FUNCTION_BLOCK FINAL FB_Cylinder EXTENDS FB_EventLogger 
VAR_INPUT
	Energized						: BOOL;							//Optional Energize Input
END_VAR                                                     		
VAR_IN_OUT                                                  		
	Control							: ST_System;					//Machine Control Instance
END_VAR                                                     		
VAR                                                         		
	_AutoExtend						: BOOL;							//Automated Extend Signal
	_AutoRetract					: BOOL;							//Automated Retract Signal
	_ManExtend						: BOOL;							//Screen Selection
	_ManRetract						: BOOL;							//Screen Selection
	_ManOff							: BOOL;							//Screen Selection
	_ForceExtend					: BOOL;							//Screen Selection
	_ForceRetract					: BOOL;							//Screen Selection
	_ForceOff						: BOOL;							//Screen Selection
	_CycleEnable					: BOOL;							//Cylinder Cylce Enable
	_ExtendReed1		AT %I*		: BOOL;							//Cylinder Extend Reed 1
	_ExtendReed2		AT %I*		: BOOL;							//Cylinder Extend Reed 2
	_ExtendReed3		AT %I*		: BOOL;							//Cylinder Extend Reed 3
	_ExtendReed4		AT %I*		: BOOL;							//Cylinder Extend Reed 4
	_RetractReed1		AT %I*		: BOOL;							//Cylinder Retract Reed 1
	_RetractReed2		AT %I*		: BOOL;							//Cylinder Retract Reed 2
	_RetractReed3		AT %I*		: BOOL;							//Cylinder Retract Reed 3
	_RetractReed4		AT %I*		: BOOL;							//Cylinder Retract Reed 4
	_DualSolenoid					: BOOL;							//Configured as a dual Solenoid Device
	_SingleSolenoidNormal			: BOOL;							//Configured as a Signal Solenoid Extend Device (Default)	
	_SingleSolenoidReverse			: BOOL;							//Configured as a Signal Solenoid Retract Device
	_CountsReset					: BOOL;							//Cycle Counts Reset
	_CycleExtend					: BOOL;							//Cylinder Cycle Extend
	_CycleRetract					: BOOL;							//Cylinder Cycle Retract
	_ExtendSolOnTime_ET				: REAL;							//Time Extend Solenoid Has Been Energised
	_ExtendSolOffTime_ET			: REAL;							//Time Since Extend Solenoid was Last Energised
	_RetractSolOnTime_ET			: REAL;							//Time Retract Solenoid Has Been Energised
	_RetractSolOffTime_ET			: REAL;							//Time Since Retract Solenoid was Last Energised
	_ExtendTime_ET					: REAL;							//Time Cylinder has been Extended
	_RetractTime_ET					: REAL;							//Time Cylinder has been Retracted
	_CycleExtTime_ET				: REAL;							//Cylinder Cycle Extend Accumulated Time
	_CycleRetTime_ET				: REAL;							//Cylinder Cycle Retract Accumulated Time
	_ExtendReed						: BOOL;							//All cylinder extend reeds have been made
	_RetractReed					: BOOL;							//All cylinder retract reeds have been made
	_ReedFaultCount					: SINT;							//Count for type of reed fault
	_ExtendSol				AT %Q*	: BOOL;							//Physical output for extend solenoid
	_RetractSol				AT %Q*	: BOOL;							//Physical output for retract solenoid
	_ExtendFault					: BOOL;							//Fault for cylinder extend
	_RetractFault					: BOOL;							//Fault for cylinder retract
	_ReedFault						: BOOL;							//Fault for reed
	_ReedFaultTime_ET				: REAL;							//Reed fault elapsed time
	_ExFaultTime_ET					: REAL;							//Extend fault elapsed time
	_RtFaultTime_ET					: REAL;							//Retract fault elapsed time
	_Alarm							: BOOL;							//Device Alarm
	_Warning						: BOOL;							//Device Warning
	_AlarmNum						: DINT;							//Device Alarm Number
	_WarningNum						: DINT;							//Device Warning Number
	_Mute_Retract					: BOOL;							//Mute Retract Alarm
	_Mute_Extend					: BOOL;							//Mute Extend Alarm
	_extendReedUsed1				: BOOL;                 	
	_extendReedUsed2				: BOOL;                 	
	_extendReedUsed3				: BOOL;                 	
	_extendReedUsed4				: BOOL;                 	
	_retractReedUsed1				: BOOL;
	_retractReedUsed2				: BOOL;
	_retractReedUsed3				: BOOL;
	_retractReedUsed4				: BOOL;
	_R_Trig							: ARRAY[0..19] OF R_TRIG;		//Private Rising Edge Triggers
END_VAR
VAR PERSISTENT
	_Name							: STRING[15];					//Name for HMI
	_Description					: STRING[40];					//Description for HMI
	_AlarmMute						: BOOL;							//Alarm Mute
	_TypeCfg						: E_CylinderTypeConfig;			//Type Selection from Screen
	_ExtendReedsUsed				: WORD;							//Data Word for Number of Extend Reeds used
	_RetractReedsUsed				: WORD;							//Data Word for Number of Retract Reeds used
	_ExtendCount					: REAL;							//Total number of cylinder extends
	_RetractCount					: REAL;							//Total number of cylinder retracts
	_ReedFaultTime_PT				: REAL;							//Reed Fault Preset Time
	_ExFaultTime_PT					: REAL;							//Extend Fault Preset Time
	_RtFaultTime_PT					: REAL;							//Retract Fault Preset Time
	_CycleExtTime_PT				: REAL;							//Cylinder Cycle Extend Time Preset
	_CycleRetTime_PT				: REAL;							//Cylinder Cycle Retract Time Preset
	_Variables						: ARRAY [0..9] OF ST_Variable;	//Device Associated Varibles Array	
END_VAR

M_AlarmMonitor();
M_WarningMonitor();
M_CountsReset();
M_UnlatchManuals();
M_TypeConfig();
M_TestCycle();
M_Extend();
M_Retract();
M_ExtendFault();
M_RetractFault();
M_ReedFault();
M_ReedControl();

{attribute 'monitoring' := 'variable'}
PROPERTY PUBLIC Alarm : Bool
GET
Alarm := _Alarm;
END_GET
END_PROPERTY

{attribute 'monitoring' := 'variable'}
PROPERTY PUBLIC AlarmMute : BOOL
SET
AlarmMute := _AlarmMute;
END_SET
END_PROPERTY

{attribute 'monitoring' := 'variable'}
PROPERTY PUBLIC AutoExtend : Bool
SET
_AutoExtend:= AutoExtend;
END_SET
END_PROPERTY

{attribute 'monitoring' := 'variable'}
PROPERTY PUBLIC AutoRetract : Bool
SET
_AutoRetract:= AutoRetract;
END_SET
END_PROPERTY

{attribute 'monitoring' := 'variable'}
PROPERTY PUBLIC CycleExtTime_PT : real
GET
CycleExtTime_PT := _CycleExtTime_PT;
END_GET
SET
_CycleExtTime_PT := CycleExtTime_PT;
END_SET
END_PROPERTY

{attribute 'monitoring' := 'variable'}
PROPERTY PUBLIC CycleRetTime_PT : real
GET
CycleRetTime_PT := _CycleRetTime_PT;
END_GET
SET
_CycleRetTime_PT := CycleRetTime_PT;
END_SET
END_PROPERTY

{attribute 'monitoring' := 'variable'}
PROPERTY PUBLIC Description : String[40]
GET
Description := _Description;
END_GET
SET
_Description := Description;
END_SET
END_PROPERTY

{attribute 'monitoring' := 'variable'}
PROPERTY PUBLIC ExFaultTime_ET : real
GET
ExFaultTime_ET := _ExFaultTime_ET;
END_GET
END_PROPERTY

{attribute 'monitoring' := 'variable'}
PROPERTY PUBLIC ExFaultTime_PT : real
GET
ExFaultTime_PT := _ExFaultTime_PT;
END_GET
SET
_ExFaultTime_PT := ExFaultTime_PT;
END_SET
END_PROPERTY

{attribute 'monitoring' := 'variable'}
PROPERTY PUBLIC ExtendReed : Bool
GET
ExtendReed := _ExtendReed;
END_GET
END_PROPERTY

{attribute 'monitoring' := 'variable'}
PROPERTY PUBLIC ExtendReed1 : Bool
GET
ExtendReed1 := _ExtendReed;
END_GET
SET // PUBLIC
_ExtendReed1 := ExtendReed1;
END_SET
END_PROPERTY

{attribute 'monitoring' := 'variable'}
PROPERTY PUBLIC ExtendSol : Bool
GET
ExtendSol := _ExtendSol;
END_GET
END_PROPERTY

{attribute 'monitoring' := 'variable'}
PROPERTY PUBLIC ForceExtend : Bool
GET
ForceExtend := _ForceExtend;
END_GET
SET
_ForceExtend := ForceExtend;
END_SET
END_PROPERTY

{attribute 'monitoring' := 'variable'}
PROPERTY PUBLIC ForceRetract : Bool
GET
ForceRetract := _ForceRetract;
END_GET
SET
_ForceRetract := ForceRetract;
END_SET
END_PROPERTY

METHOD PRIVATE M_AlarmMonitor
VAR_INPUT
END_VAR
VAR_INST // added by the converter: edge detectors and wires of the graphical bodies
    _w1, _w2, _w3, _w4, _w5 : BOOL;
END_VAR
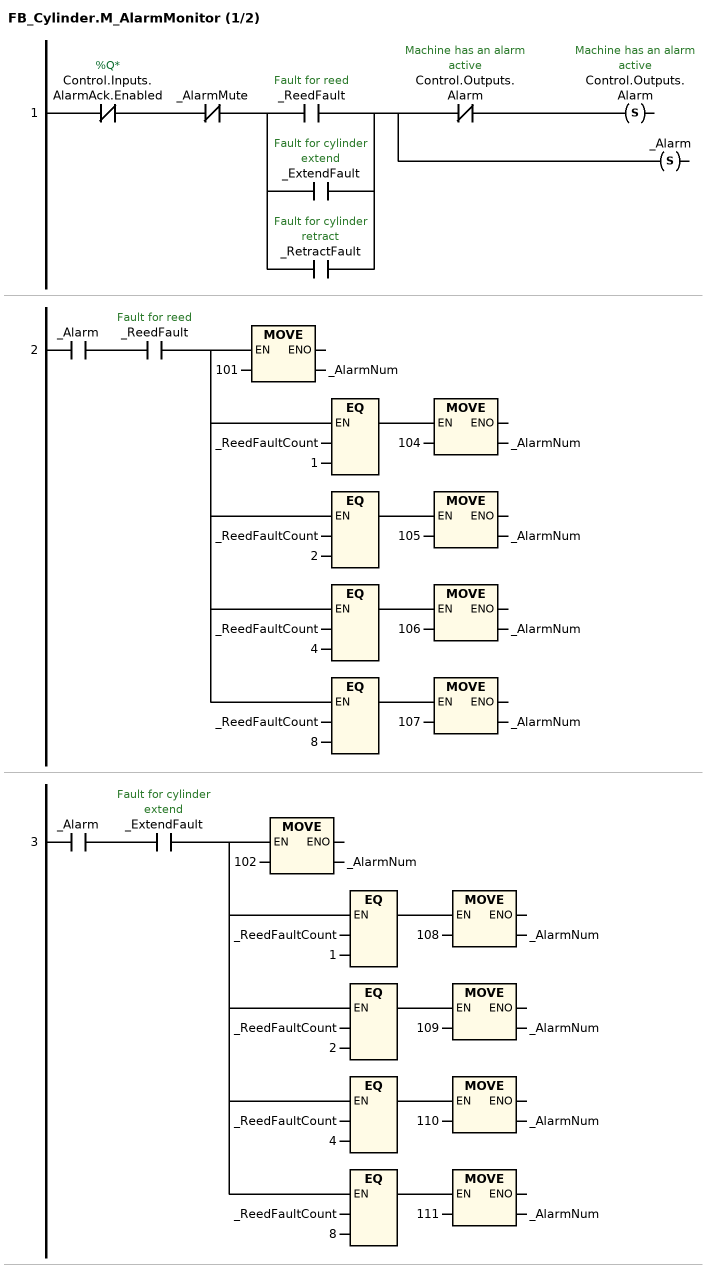
// NETWORK 1
//   Control.Inputs.AlarmAck.Enabled: AT %Q*
//   _ReedFault: Fault for reed
//   _ExtendFault: Fault for cylinder extend
//   _RetractFault: Fault for cylinder retract
//   Control.Outputs.Alarm: Machine has an alarm active
_w1 := NOT Control.Inputs.AlarmAck.Enabled AND NOT _AlarmMute AND (_ReedFault OR _ExtendFault OR _RetractFault);
Control.Outputs.Alarm S= _w1 AND NOT Control.Outputs.Alarm;
_Alarm S= _w1;

// NETWORK 2
//   _ReedFault: Fault for reed
//   _ReedFaultCount: Count for type of reed fault
_w2 := _Alarm AND _ReedFault;
IF _w2 THEN _AlarmNum := 101; END_IF
IF _w2 AND _ReedFaultCount = 1 THEN _AlarmNum := 104; END_IF
IF _w2 AND _ReedFaultCount = 2 THEN _AlarmNum := 105; END_IF
IF _w2 AND _ReedFaultCount = 4 THEN _AlarmNum := 106; END_IF
IF _w2 AND _ReedFaultCount = 8 THEN _AlarmNum := 107; END_IF

// NETWORK 3
//   _ExtendFault: Fault for cylinder extend
//   _ReedFaultCount: Count for type of reed fault
_w3 := _Alarm AND _ExtendFault;
IF _w3 THEN _AlarmNum := 102; END_IF
IF _w3 AND _ReedFaultCount = 1 THEN _AlarmNum := 108; END_IF
IF _w3 AND _ReedFaultCount = 2 THEN _AlarmNum := 109; END_IF
IF _w3 AND _ReedFaultCount = 4 THEN _AlarmNum := 110; END_IF
IF _w3 AND _ReedFaultCount = 8 THEN _AlarmNum := 111; END_IF

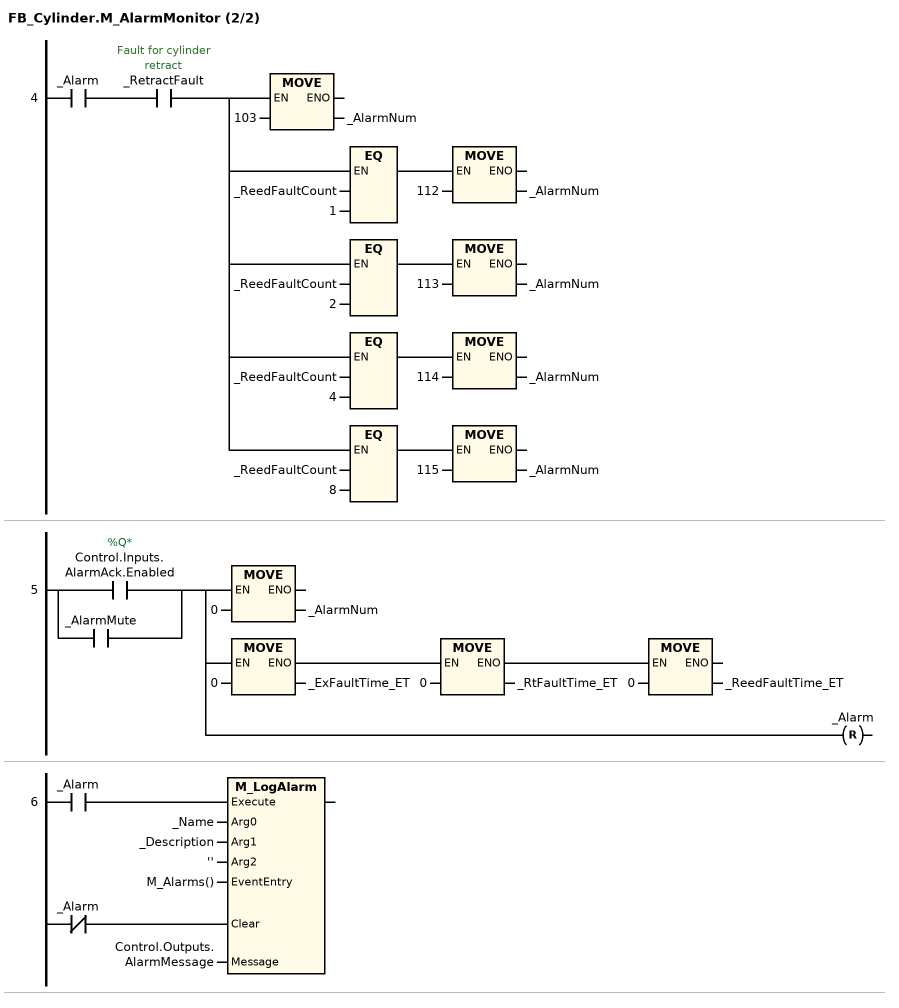
// NETWORK 4
//   _RetractFault: Fault for cylinder retract
//   _ReedFaultCount: Count for type of reed fault
_w4 := _Alarm AND _RetractFault;
IF _w4 THEN _AlarmNum := 103; END_IF
IF _w4 AND _ReedFaultCount = 1 THEN _AlarmNum := 112; END_IF
IF _w4 AND _ReedFaultCount = 2 THEN _AlarmNum := 113; END_IF
IF _w4 AND _ReedFaultCount = 4 THEN _AlarmNum := 114; END_IF
IF _w4 AND _ReedFaultCount = 8 THEN _AlarmNum := 115; END_IF

// NETWORK 5
//   Control.Inputs.AlarmAck.Enabled: AT %Q*
//   _ExFaultTime_ET: Extend fault elapsed time
//   _RtFaultTime_ET: Retract fault elapsed time
//   _ReedFaultTime_ET: Reed fault elapsed time
_w5 := Control.Inputs.AlarmAck.Enabled OR _AlarmMute;
IF _w5 THEN _AlarmNum := 0; END_IF
IF _w5 THEN _ExFaultTime_ET := 0; END_IF
IF _w5 THEN _RtFaultTime_ET := 0; END_IF
IF _w5 THEN _ReedFaultTime_ET := 0; END_IF
_Alarm R= _w5;

// NETWORK 6
M_LogAlarm(Execute := _Alarm, Arg0 := _Name, Arg1 := _Description, Arg2 := '', EventEntry := M_Alarms(), Clear := NOT _Alarm, Message := Control.Outputs.AlarmMessage);
END_METHOD

METHOD PRIVATE M_Alarms : TcEventEntry
VAR_INPUT
END_VAR
CASE _AlarmNum OF
	101: M_Alarms:= TC_Events.TcCylinder.A_101;//Reed Alarm
	102: M_Alarms:= TC_Events.TcCylinder.A_102;//Extend Alarm	
	103: M_Alarms:= TC_Events.TcCylinder.A_103;//Retract Alarm
	104: M_Alarms:= TC_Events.TcCylinder.A_104;//Reed A Alarm
	105: M_Alarms:= TC_Events.TcCylinder.A_105;//Reed B Alarm		
	106: M_Alarms:= TC_Events.TcCylinder.A_106;//Reed C Alarm		
	107: M_Alarms:= TC_Events.TcCylinder.A_107;//Reed D Alarm
	108: M_Alarms:= TC_Events.TcCylinder.A_108;//Extend Reed A Alarm
	109: M_Alarms:= TC_Events.TcCylinder.A_109;//Extend Reed B Alarm
	110: M_Alarms:= TC_Events.TcCylinder.A_110;//Extend Reed C Alarm	
	111: M_Alarms:= TC_Events.TcCylinder.A_111;//Extend Reed D Alarm		
	112: M_Alarms:= TC_Events.TcCylinder.A_112;//Retract Reed A Alarm	
	113: M_Alarms:= TC_Events.TcCylinder.A_113;//Retract Reed B Alarm	
	114: M_Alarms:= TC_Events.TcCylinder.A_114;//Retract Reed C Alarm
	115: M_Alarms:= TC_Events.TcCylinder.A_115;//Retract Reed D Alarm
ELSE
	M_Alarms:= TC_Events.TcCylinder.A_Undefined;
END_CASE
END_METHOD

METHOD PRIVATE M_CountsReset
VAR_INPUT
END_VAR
IF _CountsReset THEN
	_ExtendCount := 0;
	_RetractCount := 0;
END_IF
END_METHOD

METHOD PRIVATE M_Extend
VAR_INPUT
END_VAR
VAR_INST // added by the converter: edge detectors and wires of the graphical bodies
    _w1, _w2 : BOOL;
END_VAR
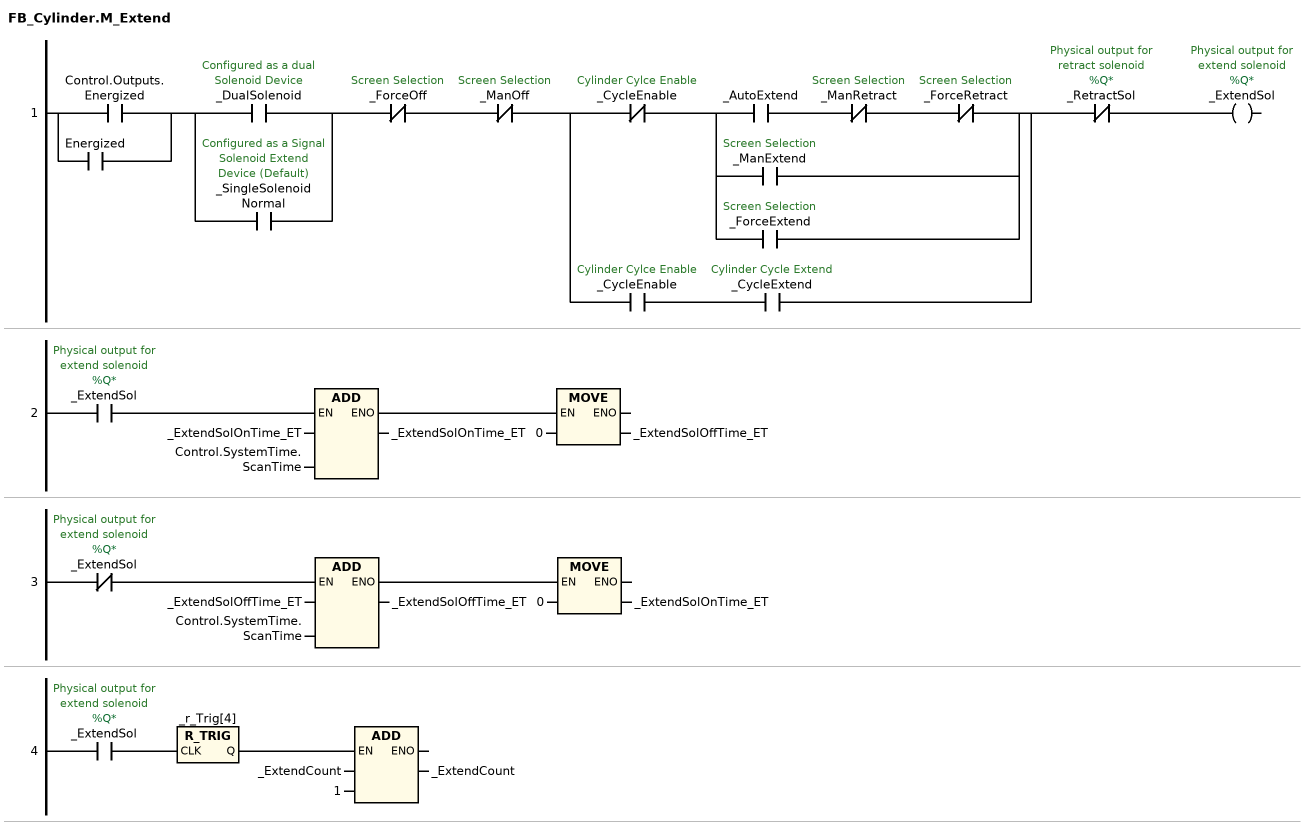
// NETWORK 1
//   _DualSolenoid: Configured as a dual Solenoid Device
//   _SingleSolenoidNormal: Configured as a Signal Solenoid Extend Device (Default)
//   _ForceOff: Screen Selection
//   _ManOff: Screen Selection
//   _CycleEnable: Cylinder Cylce Enable
//   _ManRetract: Screen Selection
//   _ForceRetract: Screen Selection
//   _ManExtend: Screen Selection
//   _ForceExtend: Screen Selection
//   _CycleExtend: Cylinder Cycle Extend
//   _RetractSol: Physical output for retract solenoid | AT %Q*
//   _ExtendSol: Physical output for extend solenoid | AT %Q*
_ExtendSol := (Control.Outputs.Energized OR Energized) AND (_DualSolenoid OR _SingleSolenoidNormal) AND NOT _ForceOff AND NOT _ManOff AND (NOT _CycleEnable AND (_AutoExtend AND NOT _ManRetract AND NOT _ForceRetract OR _ManExtend OR _ForceExtend) OR _CycleEnable AND _CycleExtend) AND NOT _RetractSol;

// NETWORK 2
//   _ExtendSol: Physical output for extend solenoid | AT %Q*
//   _ExtendSolOnTime_ET: Time Extend Solenoid Has Been Energised
//   Control.SystemTime.ScanTime: Last scan time (Seconds)
//   _ExtendSolOffTime_ET: Time Since Extend Solenoid was Last Energised
_w1 := _ExtendSol;
IF _w1 THEN _ExtendSolOnTime_ET := _ExtendSolOnTime_ET + Control.SystemTime.ScanTime; END_IF
IF _w1 THEN _ExtendSolOffTime_ET := 0; END_IF

// NETWORK 3
//   _ExtendSol: Physical output for extend solenoid | AT %Q*
//   _ExtendSolOffTime_ET: Time Since Extend Solenoid was Last Energised
//   Control.SystemTime.ScanTime: Last scan time (Seconds)
//   _ExtendSolOnTime_ET: Time Extend Solenoid Has Been Energised
_w2 := NOT _ExtendSol;
IF _w2 THEN _ExtendSolOffTime_ET := _ExtendSolOffTime_ET + Control.SystemTime.ScanTime; END_IF
IF _w2 THEN _ExtendSolOnTime_ET := 0; END_IF

// NETWORK 4
//   _ExtendSol: Physical output for extend solenoid | AT %Q*
//   _ExtendCount: Total number of cylinder extends
_r_Trig[4](CLK := _ExtendSol); // R_TRIG
IF _r_Trig[4].Q THEN _ExtendCount := _ExtendCount + 1; END_IF
END_METHOD

METHOD PRIVATE M_ExtendFault
VAR_INPUT
END_VAR
VAR_INST
	_extending					: BOOL;
	_extendReedFault_Q			: BOOL;
	_extendReedFaultArray		: ARRAY[0..4] OF BOOL;
END_VAR
VAR_INST // added by the converter: edge detectors and wires of the graphical bodies
    _w1, _w2, _w3, _w4, _w5 : BOOL;
END_VAR
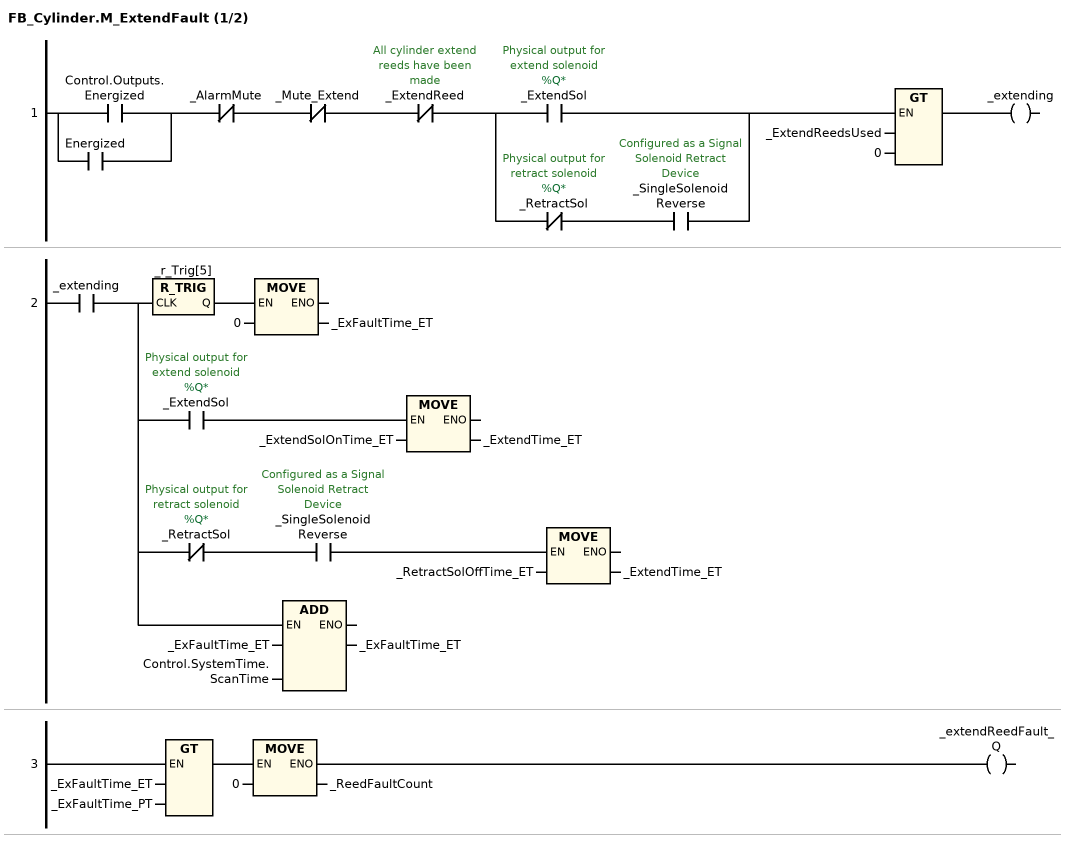
// NETWORK 1
//   _ExtendReed: All cylinder extend reeds have been made
//   _ExtendSol: Physical output for extend solenoid | AT %Q*
//   _RetractSol: Physical output for retract solenoid | AT %Q*
//   _SingleSolenoidReverse: Configured as a Signal Solenoid Retract Device
//   _ExtendReedsUsed: Data Word for Number of Extend Reeds used
_extending := (Control.Outputs.Energized OR Energized) AND NOT _AlarmMute AND NOT _Mute_Extend AND NOT _ExtendReed AND (_ExtendSol OR NOT _RetractSol AND _SingleSolenoidReverse) AND _ExtendReedsUsed > 0;

// NETWORK 2
//   _ExFaultTime_ET: Extend fault elapsed time
//   _ExtendSol: Physical output for extend solenoid | AT %Q*
//   _ExtendSolOnTime_ET: Time Extend Solenoid Has Been Energised
//   _ExtendTime_ET: Time Cylinder has been Extended
//   _RetractSol: Physical output for retract solenoid | AT %Q*
//   _SingleSolenoidReverse: Configured as a Signal Solenoid Retract Device
//   _RetractSolOffTime_ET: Time Since Retract Solenoid was Last Energised
//   Control.SystemTime.ScanTime: Last scan time (Seconds)
_r_Trig[5](CLK := _extending); // R_TRIG
IF _r_Trig[5].Q THEN _ExFaultTime_ET := 0; END_IF
IF _extending AND _ExtendSol THEN _ExtendTime_ET := _ExtendSolOnTime_ET; END_IF
IF _extending AND NOT _RetractSol AND _SingleSolenoidReverse THEN _ExtendTime_ET := _RetractSolOffTime_ET; END_IF
IF _extending THEN _ExFaultTime_ET := _ExFaultTime_ET + Control.SystemTime.ScanTime; END_IF

// NETWORK 3
//   _ExFaultTime_ET: Extend fault elapsed time
//   _ReedFaultCount: Count for type of reed fault
_w1 := _ExFaultTime_ET > _ExFaultTime_PT;
IF _w1 THEN _ReedFaultCount := 0; END_IF
_extendReedFault_Q := _w1;

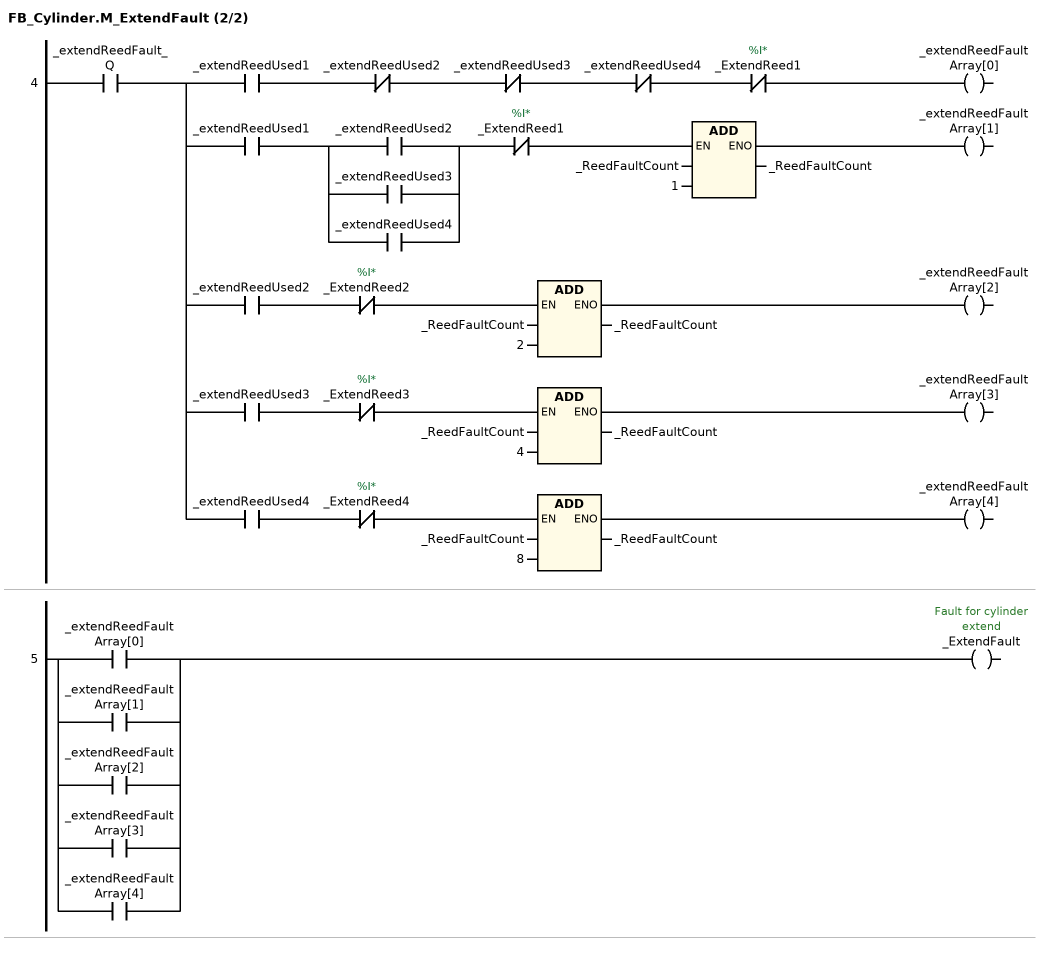
// NETWORK 4
//   _ExtendReed1: AT %I*
//   _ReedFaultCount: Count for type of reed fault
//   _ExtendReed2: AT %I*
//   _ExtendReed3: AT %I*
//   _ExtendReed4: AT %I*
_extendReedFaultArray[0] := _extendReedFault_Q AND _extendReedUsed1 AND NOT _extendReedUsed2 AND NOT _extendReedUsed3 AND NOT _extendReedUsed4 AND NOT _ExtendReed1;
_w2 := _extendReedFault_Q AND _extendReedUsed1 AND (_extendReedUsed2 OR _extendReedUsed3 OR _extendReedUsed4) AND NOT _ExtendReed1;
IF _w2 THEN _ReedFaultCount := _ReedFaultCount + 1; END_IF
_extendReedFaultArray[1] := _w2;
_w3 := _extendReedFault_Q AND _extendReedUsed2 AND NOT _ExtendReed2;
IF _w3 THEN _ReedFaultCount := _ReedFaultCount + 2; END_IF
_extendReedFaultArray[2] := _w3;
_w4 := _extendReedFault_Q AND _extendReedUsed3 AND NOT _ExtendReed3;
IF _w4 THEN _ReedFaultCount := _ReedFaultCount + 4; END_IF
_extendReedFaultArray[3] := _w4;
_w5 := _extendReedFault_Q AND _extendReedUsed4 AND NOT _ExtendReed4;
IF _w5 THEN _ReedFaultCount := _ReedFaultCount + 8; END_IF
_extendReedFaultArray[4] := _w5;

// NETWORK 5
//   _ExtendFault: Fault for cylinder extend
_ExtendFault := _extendReedFaultArray[0] OR _extendReedFaultArray[1] OR _extendReedFaultArray[2] OR _extendReedFaultArray[3] OR _extendReedFaultArray[4];
END_METHOD

METHOD PRIVATE M_ReedControl
VAR_INPUT
END_VAR
VAR_INST
END_VAR
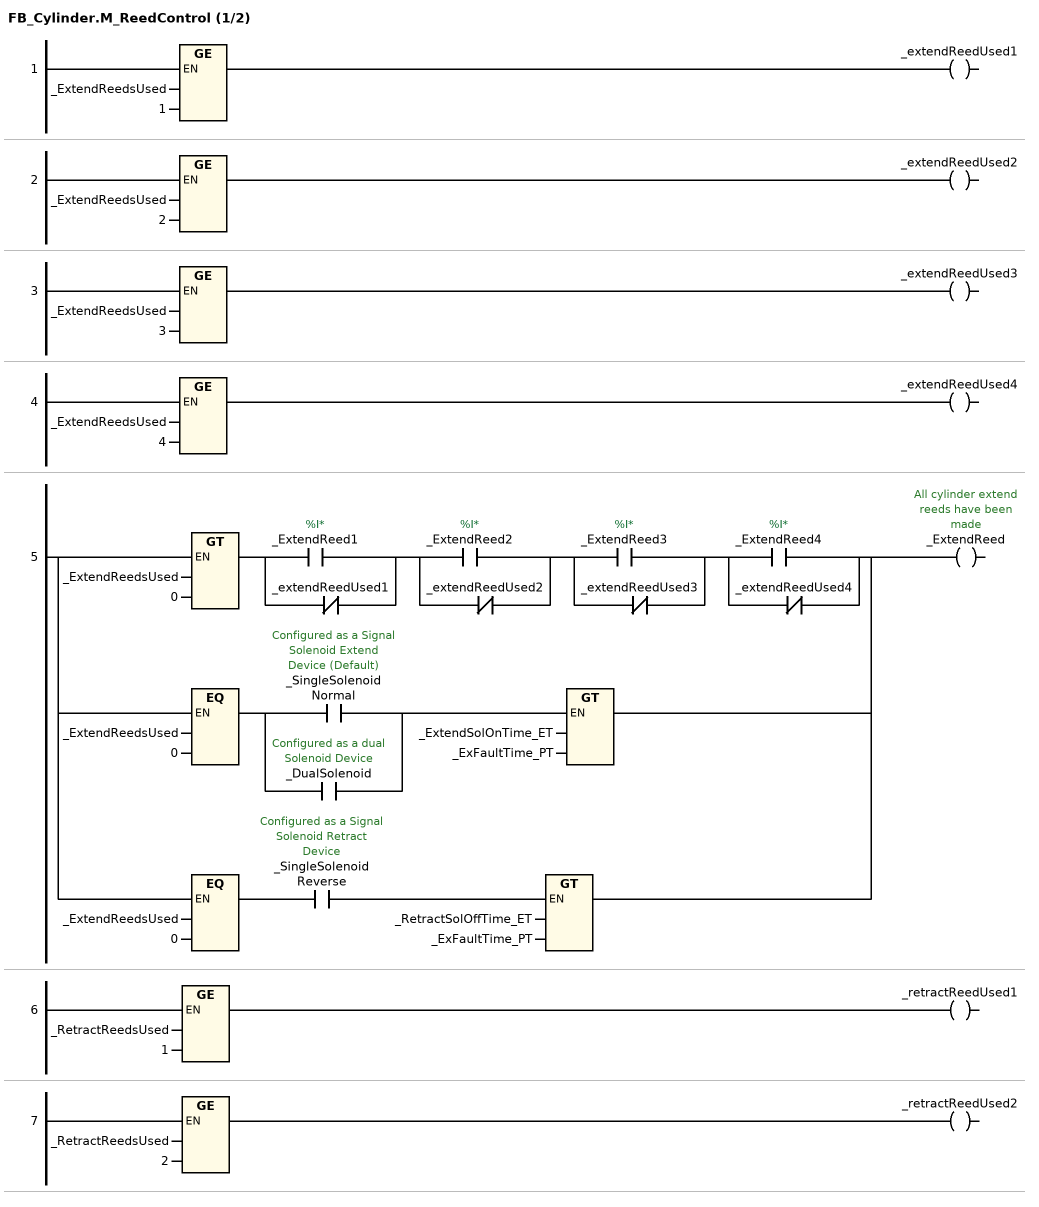
// NETWORK 1
//   _ExtendReedsUsed: Data Word for Number of Extend Reeds used
_extendReedUsed1 := _ExtendReedsUsed >= 1;

// NETWORK 2
//   _ExtendReedsUsed: Data Word for Number of Extend Reeds used
_extendReedUsed2 := _ExtendReedsUsed >= 2;

// NETWORK 3
//   _ExtendReedsUsed: Data Word for Number of Extend Reeds used
_extendReedUsed3 := _ExtendReedsUsed >= 3;

// NETWORK 4
//   _ExtendReedsUsed: Data Word for Number of Extend Reeds used
_extendReedUsed4 := _ExtendReedsUsed >= 4;

// NETWORK 5
//   _ExtendReedsUsed: Data Word for Number of Extend Reeds used
//   _ExtendReed1: AT %I*
//   _ExtendReed2: AT %I*
//   _ExtendReed3: AT %I*
//   _ExtendReed4: AT %I*
//   _SingleSolenoidNormal: Configured as a Signal Solenoid Extend Device (Default)
//   _DualSolenoid: Configured as a dual Solenoid Device
//   _ExtendSolOnTime_ET: Time Extend Solenoid Has Been Energised
//   _SingleSolenoidReverse: Configured as a Signal Solenoid Retract Device
//   _RetractSolOffTime_ET: Time Since Retract Solenoid was Last Energised
//   _ExtendReed: All cylinder extend reeds have been made
_ExtendReed := _ExtendReedsUsed > 0 AND (_ExtendReed1 OR NOT _extendReedUsed1) AND (_ExtendReed2 OR NOT _extendReedUsed2) AND (_ExtendReed3 OR NOT _extendReedUsed3) AND (_ExtendReed4 OR NOT _extendReedUsed4) OR _ExtendReedsUsed = 0 AND (_SingleSolenoidNormal OR _DualSolenoid) AND _ExtendSolOnTime_ET > _ExFaultTime_PT OR _ExtendReedsUsed = 0 AND _SingleSolenoidReverse AND _RetractSolOffTime_ET > _ExFaultTime_PT;

// NETWORK 6
//   _RetractReedsUsed: Data Word for Number of Retract Reeds used
_retractReedUsed1 := _RetractReedsUsed >= 1;

// NETWORK 7
//   _RetractReedsUsed: Data Word for Number of Retract Reeds used
_retractReedUsed2 := _RetractReedsUsed >= 2;

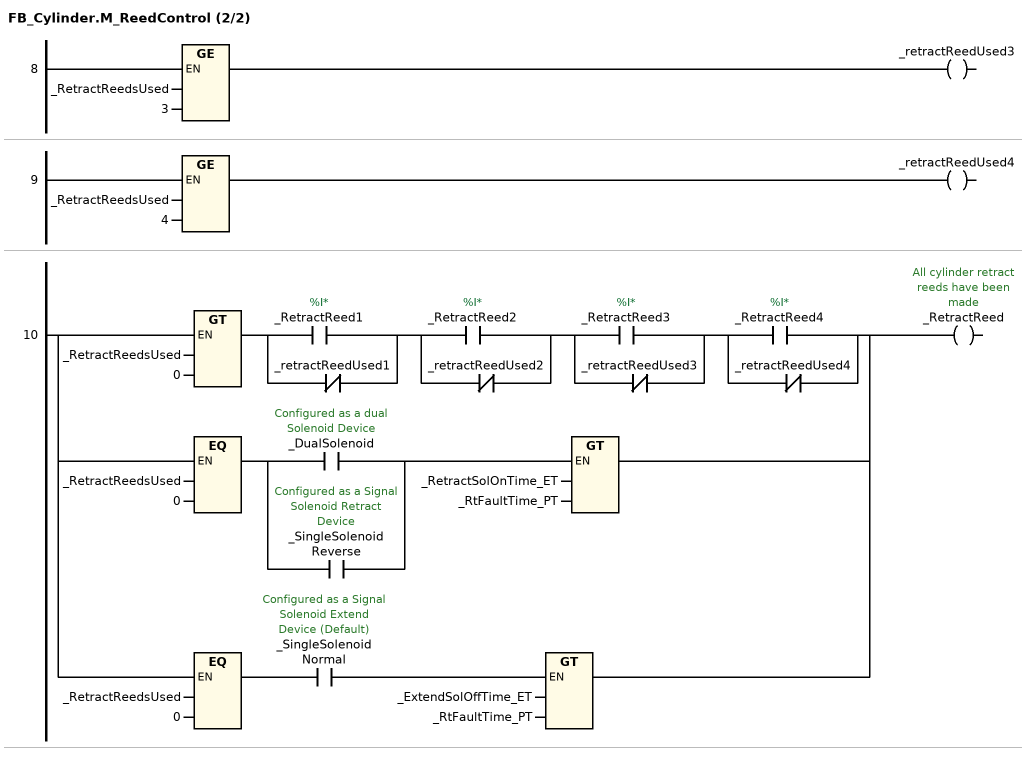
// NETWORK 8
//   _RetractReedsUsed: Data Word for Number of Retract Reeds used
_retractReedUsed3 := _RetractReedsUsed >= 3;

// NETWORK 9
//   _RetractReedsUsed: Data Word for Number of Retract Reeds used
_retractReedUsed4 := _RetractReedsUsed >= 4;

// NETWORK 10
//   _RetractReedsUsed: Data Word for Number of Retract Reeds used
//   _RetractReed1: AT %I*
//   _RetractReed2: AT %I*
//   _RetractReed3: AT %I*
//   _RetractReed4: AT %I*
//   _DualSolenoid: Configured as a dual Solenoid Device
//   _SingleSolenoidReverse: Configured as a Signal Solenoid Retract Device
//   _RetractSolOnTime_ET: Time Retract Solenoid Has Been Energised
//   _SingleSolenoidNormal: Configured as a Signal Solenoid Extend Device (Default)
//   _ExtendSolOffTime_ET: Time Since Extend Solenoid was Last Energised
//   _RetractReed: All cylinder retract reeds have been made
_RetractReed := _RetractReedsUsed > 0 AND (_RetractReed1 OR NOT _retractReedUsed1) AND (_RetractReed2 OR NOT _retractReedUsed2) AND (_RetractReed3 OR NOT _retractReedUsed3) AND (_RetractReed4 OR NOT _retractReedUsed4) OR _RetractReedsUsed = 0 AND (_DualSolenoid OR _SingleSolenoidReverse) AND _RetractSolOnTime_ET > _RtFaultTime_PT OR _RetractReedsUsed = 0 AND _SingleSolenoidNormal AND _ExtendSolOffTime_ET > _RtFaultTime_PT;
END_METHOD

METHOD PRIVATE M_ReedFault
VAR_INPUT
END_VAR
VAR_INST
	_reedFault					: BOOL;
	_reedFault_Q				: BOOL;
	_reedFaultArray				: ARRAY[0..4] OF BOOL;
END_VAR
VAR_INST // added by the converter: edge detectors and wires of the graphical bodies
    _w1, _w2, _w3, _w4, _w5 : BOOL;
END_VAR
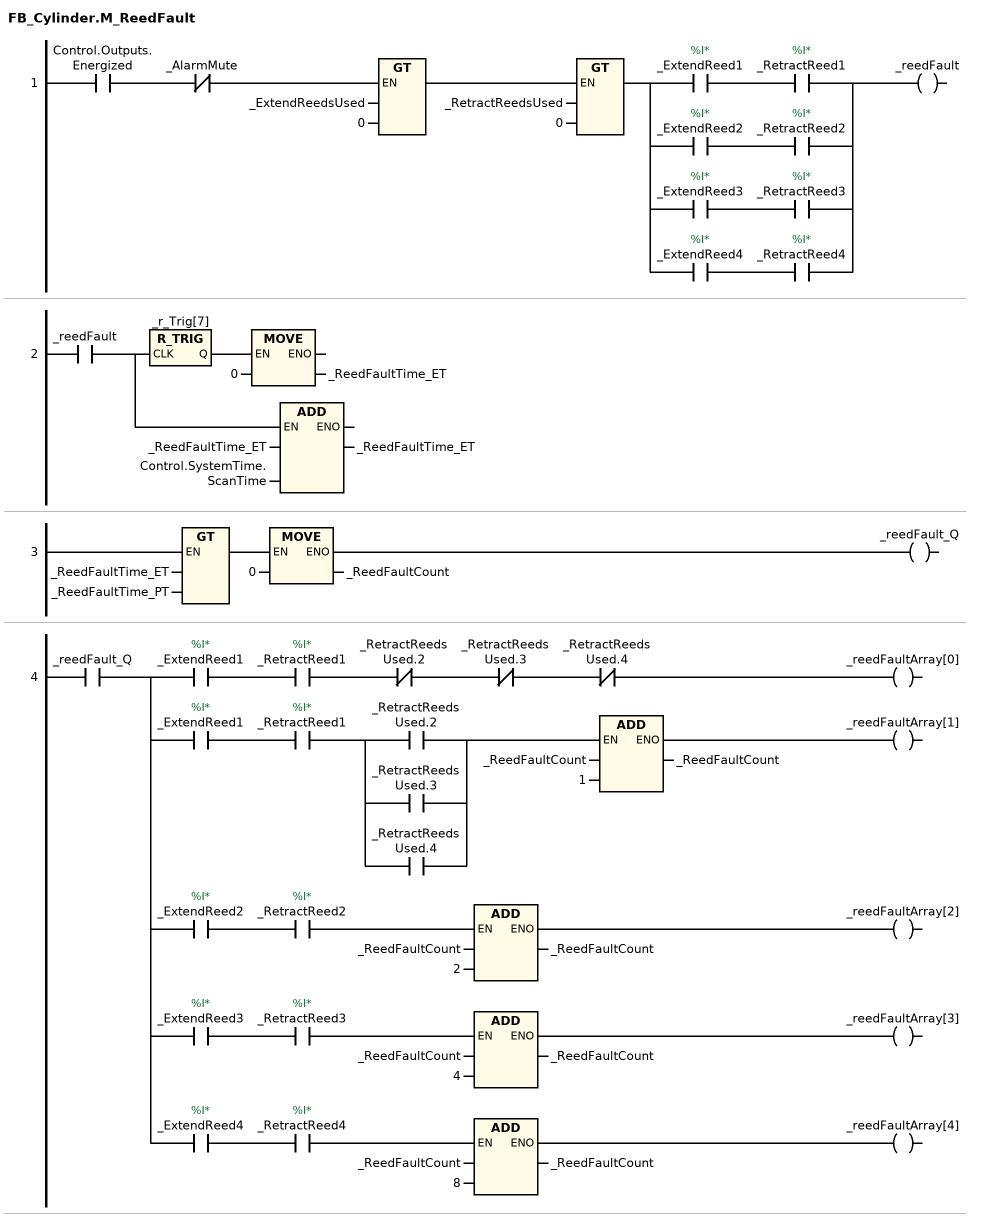
// NETWORK 1
//   _ExtendReedsUsed: Data Word for Number of Extend Reeds used
//   _RetractReedsUsed: Data Word for Number of Retract Reeds used
//   _ExtendReed1: AT %I*
//   _RetractReed1: AT %I*
//   _ExtendReed2: AT %I*
//   _RetractReed2: AT %I*
//   _ExtendReed3: AT %I*
//   _RetractReed3: AT %I*
//   _ExtendReed4: AT %I*
//   _RetractReed4: AT %I*
_reedFault := (Control.Outputs.Energized AND NOT _AlarmMute AND _ExtendReedsUsed > 0 AND _RetractReedsUsed > 0) AND (_ExtendReed1 AND _RetractReed1 OR _ExtendReed2 AND _RetractReed2 OR _ExtendReed3 AND _RetractReed3 OR _ExtendReed4 AND _RetractReed4);

// NETWORK 2
//   _ReedFaultTime_ET: Reed fault elapsed time
//   Control.SystemTime.ScanTime: Last scan time (Seconds)
_r_Trig[7](CLK := _reedFault); // R_TRIG
IF _r_Trig[7].Q THEN _ReedFaultTime_ET := 0; END_IF
IF _reedFault THEN _ReedFaultTime_ET := _ReedFaultTime_ET + Control.SystemTime.ScanTime; END_IF

// NETWORK 3
//   _ReedFaultTime_ET: Reed fault elapsed time
//   _ReedFaultCount: Count for type of reed fault
_w1 := _ReedFaultTime_ET > _ReedFaultTime_PT;
IF _w1 THEN _ReedFaultCount := 0; END_IF
_reedFault_Q := _w1;

// NETWORK 4
//   _ExtendReed1: AT %I*
//   _RetractReed1: AT %I*
//   _ReedFaultCount: Count for type of reed fault
//   _ExtendReed2: AT %I*
//   _RetractReed2: AT %I*
//   _ExtendReed3: AT %I*
//   _RetractReed3: AT %I*
//   _ExtendReed4: AT %I*
//   _RetractReed4: AT %I*
_reedFaultArray[0] := _reedFault_Q AND _ExtendReed1 AND _RetractReed1 AND NOT _RetractReedsUsed.2 AND NOT _RetractReedsUsed.3 AND NOT _RetractReedsUsed.4;
_w2 := _reedFault_Q AND _ExtendReed1 AND _RetractReed1 AND (_RetractReedsUsed.2 OR _RetractReedsUsed.3 OR _RetractReedsUsed.4);
IF _w2 THEN _ReedFaultCount := _ReedFaultCount + 1; END_IF
_reedFaultArray[1] := _w2;
_w3 := _reedFault_Q AND _ExtendReed2 AND _RetractReed2;
IF _w3 THEN _ReedFaultCount := _ReedFaultCount + 2; END_IF
_reedFaultArray[2] := _w3;
_w4 := _reedFault_Q AND _ExtendReed3 AND _RetractReed3;
IF _w4 THEN _ReedFaultCount := _ReedFaultCount + 4; END_IF
_reedFaultArray[3] := _w4;
_w5 := _reedFault_Q AND _ExtendReed4 AND _RetractReed4;
IF _w5 THEN _ReedFaultCount := _ReedFaultCount + 8; END_IF
_reedFaultArray[4] := _w5;
END_METHOD

METHOD PRIVATE M_Retract
VAR_INPUT
END_VAR
VAR_INST
END_VAR
VAR_INST // added by the converter: edge detectors and wires of the graphical bodies
    _w1, _w2 : BOOL;
END_VAR
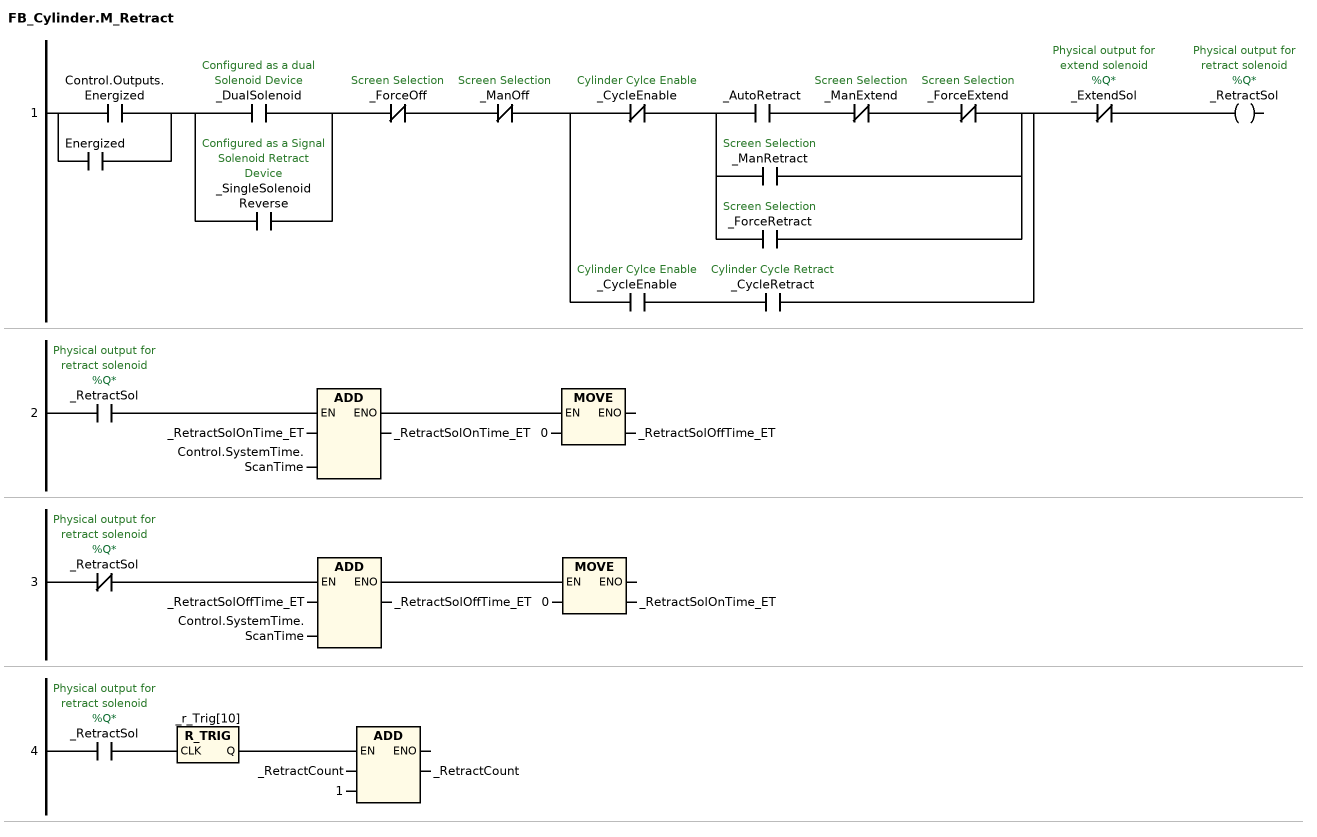
// NETWORK 1
//   _DualSolenoid: Configured as a dual Solenoid Device
//   _SingleSolenoidReverse: Configured as a Signal Solenoid Retract Device
//   _ForceOff: Screen Selection
//   _ManOff: Screen Selection
//   _CycleEnable: Cylinder Cylce Enable
//   _ManExtend: Screen Selection
//   _ForceExtend: Screen Selection
//   _ManRetract: Screen Selection
//   _ForceRetract: Screen Selection
//   _CycleRetract: Cylinder Cycle Retract
//   _ExtendSol: Physical output for extend solenoid | AT %Q*
//   _RetractSol: Physical output for retract solenoid | AT %Q*
_RetractSol := (Control.Outputs.Energized OR Energized) AND (_DualSolenoid OR _SingleSolenoidReverse) AND NOT _ForceOff AND NOT _ManOff AND (NOT _CycleEnable AND (_AutoRetract AND NOT _ManExtend AND NOT _ForceExtend OR _ManRetract OR _ForceRetract) OR _CycleEnable AND _CycleRetract) AND NOT _ExtendSol;

// NETWORK 2
//   _RetractSol: Physical output for retract solenoid | AT %Q*
//   _RetractSolOnTime_ET: Time Retract Solenoid Has Been Energised
//   Control.SystemTime.ScanTime: Last scan time (Seconds)
//   _RetractSolOffTime_ET: Time Since Retract Solenoid was Last Energised
_w1 := _RetractSol;
IF _w1 THEN _RetractSolOnTime_ET := _RetractSolOnTime_ET + Control.SystemTime.ScanTime; END_IF
IF _w1 THEN _RetractSolOffTime_ET := 0; END_IF

// NETWORK 3
//   _RetractSol: Physical output for retract solenoid | AT %Q*
//   _RetractSolOffTime_ET: Time Since Retract Solenoid was Last Energised
//   Control.SystemTime.ScanTime: Last scan time (Seconds)
//   _RetractSolOnTime_ET: Time Retract Solenoid Has Been Energised
_w2 := NOT _RetractSol;
IF _w2 THEN _RetractSolOffTime_ET := _RetractSolOffTime_ET + Control.SystemTime.ScanTime; END_IF
IF _w2 THEN _RetractSolOnTime_ET := 0; END_IF

// NETWORK 4
//   _RetractSol: Physical output for retract solenoid | AT %Q*
//   _RetractCount: Total number of cylinder retracts
_r_Trig[10](CLK := _RetractSol); // R_TRIG
IF _r_Trig[10].Q THEN _RetractCount := _RetractCount + 1; END_IF
END_METHOD

METHOD PRIVATE M_RetractFault
VAR_INPUT
END_VAR
VAR_INST
	_retracting					: BOOL;
	_retractReedFault_Q			: BOOL;
	_retractReedFaultArray		: ARRAY[0..4] OF BOOL;
END_VAR
VAR_INST // added by the converter: edge detectors and wires of the graphical bodies
    _w1, _w2, _w3, _w4, _w5 : BOOL;
END_VAR
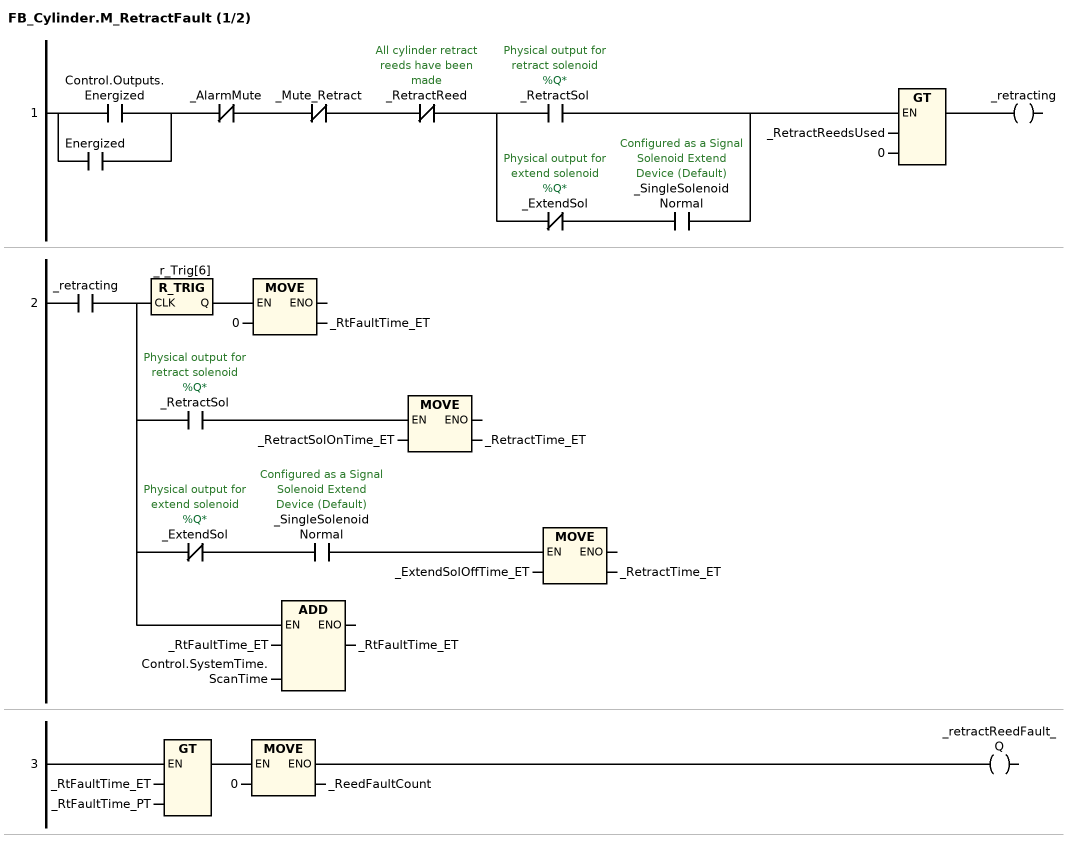
// NETWORK 1
//   _RetractReed: All cylinder retract reeds have been made
//   _RetractSol: Physical output for retract solenoid | AT %Q*
//   _ExtendSol: Physical output for extend solenoid | AT %Q*
//   _SingleSolenoidNormal: Configured as a Signal Solenoid Extend Device (Default)
//   _RetractReedsUsed: Data Word for Number of Retract Reeds used
_retracting := (Control.Outputs.Energized OR Energized) AND NOT _AlarmMute AND NOT _Mute_Retract AND NOT _RetractReed AND (_RetractSol OR NOT _ExtendSol AND _SingleSolenoidNormal) AND _RetractReedsUsed > 0;

// NETWORK 2
//   _RtFaultTime_ET: Retract fault elapsed time
//   _RetractSol: Physical output for retract solenoid | AT %Q*
//   _RetractSolOnTime_ET: Time Retract Solenoid Has Been Energised
//   _RetractTime_ET: Time Cylinder has been Retracted
//   _ExtendSol: Physical output for extend solenoid | AT %Q*
//   _SingleSolenoidNormal: Configured as a Signal Solenoid Extend Device (Default)
//   _ExtendSolOffTime_ET: Time Since Extend Solenoid was Last Energised
//   Control.SystemTime.ScanTime: Last scan time (Seconds)
_r_Trig[6](CLK := _retracting); // R_TRIG
IF _r_Trig[6].Q THEN _RtFaultTime_ET := 0; END_IF
IF _retracting AND _RetractSol THEN _RetractTime_ET := _RetractSolOnTime_ET; END_IF
IF _retracting AND NOT _ExtendSol AND _SingleSolenoidNormal THEN _RetractTime_ET := _ExtendSolOffTime_ET; END_IF
IF _retracting THEN _RtFaultTime_ET := _RtFaultTime_ET + Control.SystemTime.ScanTime; END_IF

// NETWORK 3
//   _RtFaultTime_ET: Retract fault elapsed time
//   _ReedFaultCount: Count for type of reed fault
_w1 := _RtFaultTime_ET > _RtFaultTime_PT;
IF _w1 THEN _ReedFaultCount := 0; END_IF
_retractReedFault_Q := _w1;

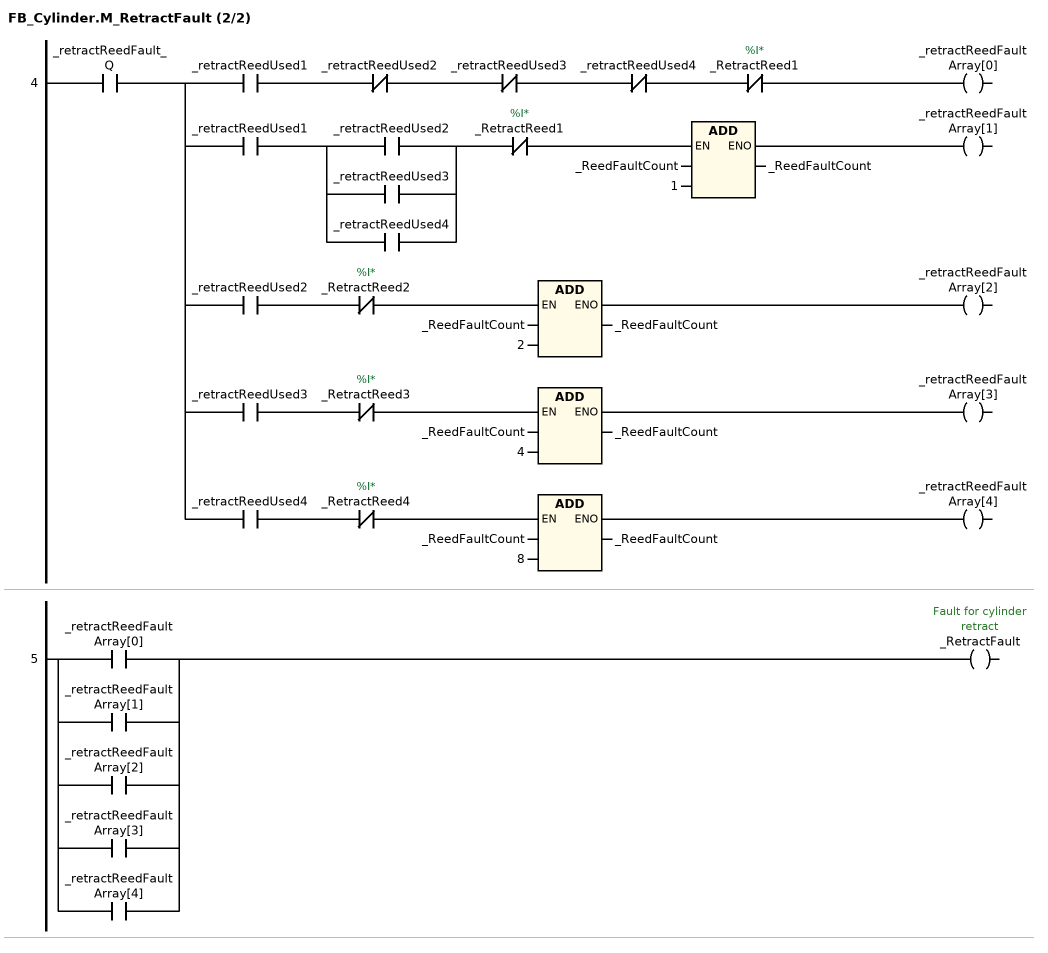
// NETWORK 4
//   _RetractReed1: AT %I*
//   _ReedFaultCount: Count for type of reed fault
//   _RetractReed2: AT %I*
//   _RetractReed3: AT %I*
//   _RetractReed4: AT %I*
_retractReedFaultArray[0] := _retractReedFault_Q AND _retractReedUsed1 AND NOT _retractReedUsed2 AND NOT _retractReedUsed3 AND NOT _retractReedUsed4 AND NOT _RetractReed1;
_w2 := _retractReedFault_Q AND _retractReedUsed1 AND (_retractReedUsed2 OR _retractReedUsed3 OR _retractReedUsed4) AND NOT _RetractReed1;
IF _w2 THEN _ReedFaultCount := _ReedFaultCount + 1; END_IF
_retractReedFaultArray[1] := _w2;
_w3 := _retractReedFault_Q AND _retractReedUsed2 AND NOT _RetractReed2;
IF _w3 THEN _ReedFaultCount := _ReedFaultCount + 2; END_IF
_retractReedFaultArray[2] := _w3;
_w4 := _retractReedFault_Q AND _retractReedUsed3 AND NOT _RetractReed3;
IF _w4 THEN _ReedFaultCount := _ReedFaultCount + 4; END_IF
_retractReedFaultArray[3] := _w4;
_w5 := _retractReedFault_Q AND _retractReedUsed4 AND NOT _RetractReed4;
IF _w5 THEN _ReedFaultCount := _ReedFaultCount + 8; END_IF
_retractReedFaultArray[4] := _w5;

// NETWORK 5
//   _RetractFault: Fault for cylinder retract
_RetractFault := _retractReedFaultArray[0] OR _retractReedFaultArray[1] OR _retractReedFaultArray[2] OR _retractReedFaultArray[3] OR _retractReedFaultArray[4];
END_METHOD

METHOD PRIVATE M_TestCycle
VAR_INPUT
END_VAR
VAR_INST
END_VAR
VAR_INST // added by the converter: edge detectors and wires of the graphical bodies
    _w1, _w2, _w3 : BOOL;
END_VAR
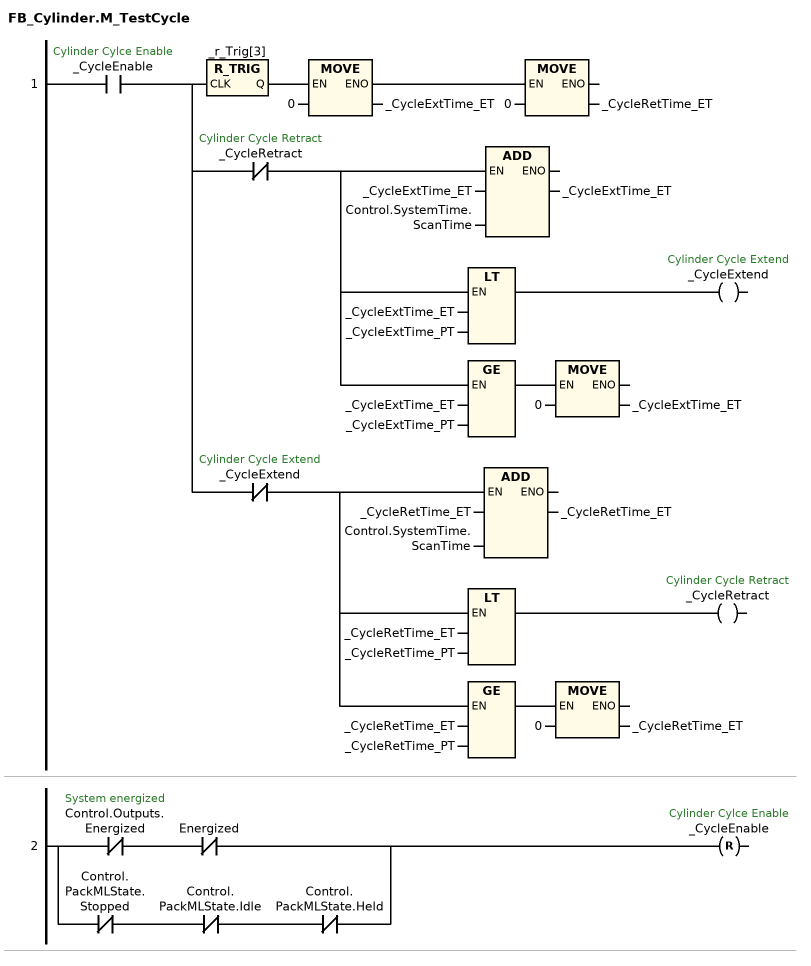
// NETWORK 1
//   _CycleEnable: Cylinder Cylce Enable
//   _CycleExtTime_ET: Cylinder Cycle Extend Accumulated Time
//   _CycleRetTime_ET: Cylinder Cycle Retract Accumulated Time
//   _CycleRetract: Cylinder Cycle Retract
//   Control.SystemTime.ScanTime: Last scan time (Seconds)
//   _CycleExtTime_PT: Cylinder Cycle Extend Time Preset
//   _CycleExtend: Cylinder Cycle Extend
//   _CycleRetTime_PT: Cylinder Cycle Retract Time Preset
_r_Trig[3](CLK := _CycleEnable); // R_TRIG
_w1 := _r_Trig[3].Q;
IF _w1 THEN _CycleExtTime_ET := 0; END_IF
IF _w1 THEN _CycleRetTime_ET := 0; END_IF
_w2 := _CycleEnable AND NOT _CycleRetract;
IF _w2 THEN _CycleExtTime_ET := _CycleExtTime_ET + Control.SystemTime.ScanTime; END_IF
_CycleExtend := _w2 AND _CycleExtTime_ET < _CycleExtTime_PT;
IF _w2 AND _CycleExtTime_ET >= _CycleExtTime_PT THEN _CycleExtTime_ET := 0; END_IF
_w3 := _CycleEnable AND NOT _CycleExtend;
IF _w3 THEN _CycleRetTime_ET := _CycleRetTime_ET + Control.SystemTime.ScanTime; END_IF
_CycleRetract := _w3 AND _CycleRetTime_ET < _CycleRetTime_PT;
IF _w3 AND _CycleRetTime_ET >= _CycleRetTime_PT THEN _CycleRetTime_ET := 0; END_IF

// NETWORK 2
//   Control.Outputs.Energized: System energized
//   _CycleEnable: Cylinder Cylce Enable
_CycleEnable R= NOT Control.Outputs.Energized AND NOT Energized OR NOT Control.PackMLState.Stopped AND NOT Control.PackMLState.Idle AND NOT Control.PackMLState.Held;
END_METHOD

METHOD PRIVATE M_TypeConfig
VAR_INPUT
END_VAR
VAR_INST
END_VAR
CASE _TypeCfg OF
	eCylinderType_SINGLE_NORMAL : 
		_SingleSolenoidNormal := TRUE;
		_SingleSolenoidReverse := FALSE;
		_DualSolenoid := FALSE;
	eCylinderType_SINGLE_REVERSE : 
		_SingleSolenoidNormal := FALSE;
		_SingleSolenoidReverse := TRUE;
		_DualSolenoid := FALSE;
	eCylinderType_DUEL : 
		_SingleSolenoidNormal := FALSE;
		_SingleSolenoidReverse := FALSE;
		_DualSolenoid := TRUE;
END_CASE
END_METHOD

METHOD PRIVATE M_UnlatchManuals
VAR_INPUT
END_VAR
VAR_INST // added by the converter: edge detectors and wires of the graphical bodies
    _rt1, _rt2, _rt3, _rt4 : R_TRIG;
END_VAR
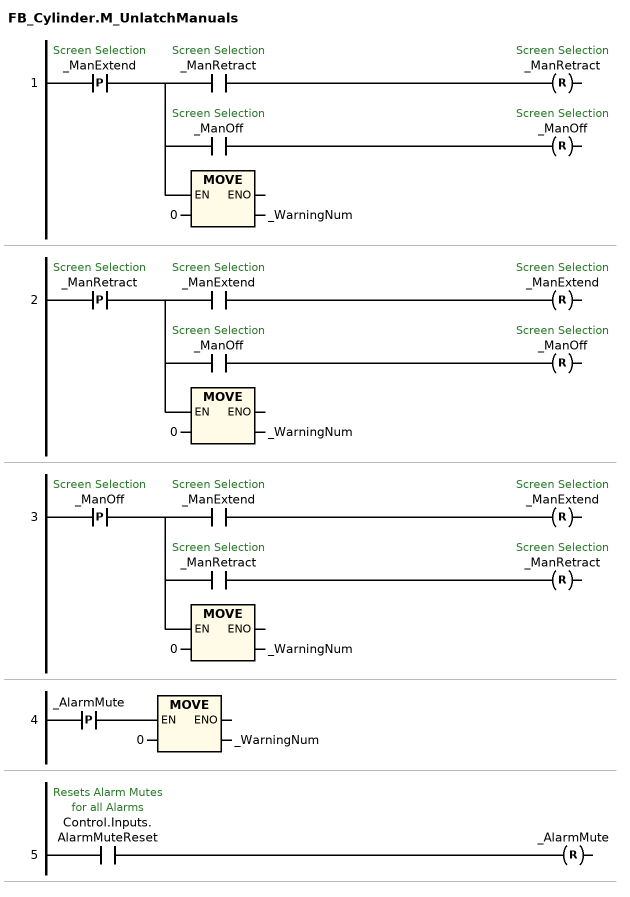
// NETWORK 1
//   _ManExtend: Screen Selection
//   _ManRetract: Screen Selection
//   _ManOff: Screen Selection
_rt1(CLK := _ManExtend);
_ManRetract R= _rt1.Q AND _ManRetract;
_ManOff R= _rt1.Q AND _ManOff;
IF _rt1.Q THEN _WarningNum := 0; END_IF

// NETWORK 2
//   _ManRetract: Screen Selection
//   _ManExtend: Screen Selection
//   _ManOff: Screen Selection
_rt2(CLK := _ManRetract);
_ManExtend R= _rt2.Q AND _ManExtend;
_ManOff R= _rt2.Q AND _ManOff;
IF _rt2.Q THEN _WarningNum := 0; END_IF

// NETWORK 3
//   _ManOff: Screen Selection
//   _ManExtend: Screen Selection
//   _ManRetract: Screen Selection
_rt3(CLK := _ManOff);
_ManExtend R= _rt3.Q AND _ManExtend;
_ManRetract R= _rt3.Q AND _ManRetract;
IF _rt3.Q THEN _WarningNum := 0; END_IF

// NETWORK 4
_rt4(CLK := _AlarmMute);
IF _rt4.Q THEN _WarningNum := 0; END_IF

// NETWORK 5
//   Control.Inputs.AlarmMuteReset: Resets Alarm Mutes for all Alarms
_AlarmMute R= Control.Inputs.AlarmMuteReset;
END_METHOD

METHOD PRIVATE M_WarningMonitor
VAR_INPUT
END_VAR
VAR_INST // added by the converter: edge detectors and wires of the graphical bodies
    _w1, _w2, _w3, _w4, _w5, _w6, _w7 : BOOL;
END_VAR
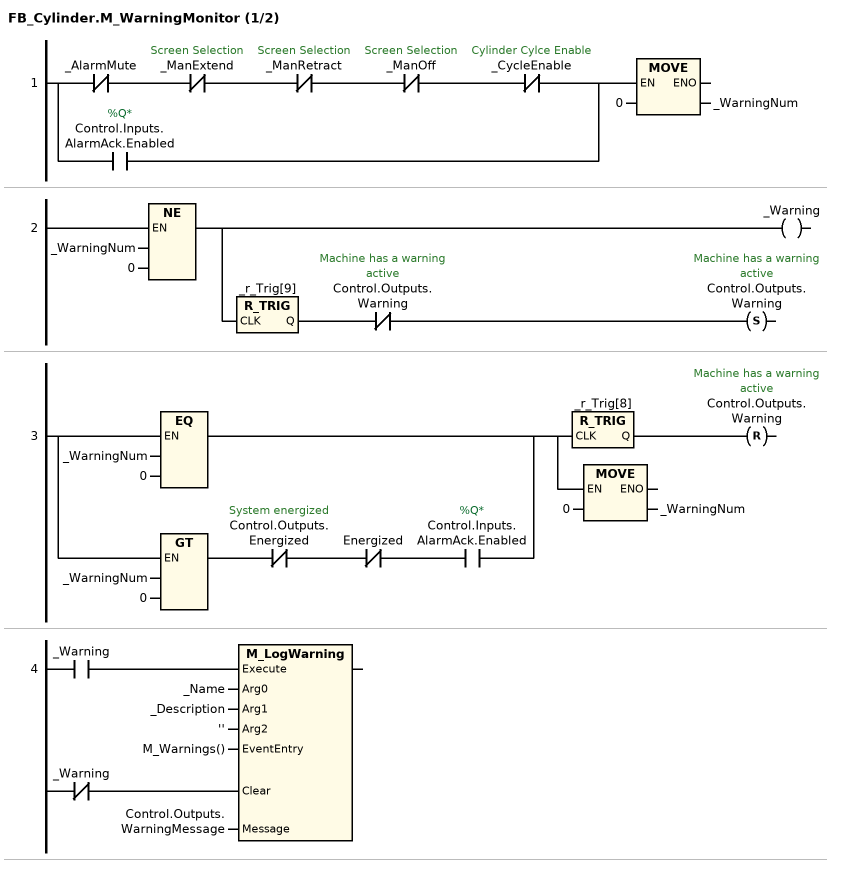
// NETWORK 1
//   _ManExtend: Screen Selection
//   _ManRetract: Screen Selection
//   _ManOff: Screen Selection
//   _CycleEnable: Cylinder Cylce Enable
//   Control.Inputs.AlarmAck.Enabled: AT %Q*
IF NOT _AlarmMute AND NOT _ManExtend AND NOT _ManRetract AND NOT _ManOff AND NOT _CycleEnable OR Control.Inputs.AlarmAck.Enabled THEN
    _WarningNum := 0;
END_IF

// NETWORK 2
//   Control.Outputs.Warning: Machine has a warning active
_w1 := _WarningNum <> 0;
_Warning := _w1;
_r_Trig[9](CLK := _w1); // R_TRIG
Control.Outputs.Warning S= _r_Trig[9].Q AND NOT Control.Outputs.Warning;

// NETWORK 3
//   Control.Outputs.Energized: System energized
//   Control.Inputs.AlarmAck.Enabled: AT %Q*
//   Control.Outputs.Warning: Machine has a warning active
_w2 := _WarningNum = 0 OR _WarningNum > 0 AND NOT Control.Outputs.Energized AND NOT Energized AND Control.Inputs.AlarmAck.Enabled;
_r_Trig[8](CLK := _w2); // R_TRIG
Control.Outputs.Warning R= _r_Trig[8].Q;
IF _w2 THEN _WarningNum := 0; END_IF

// NETWORK 4
M_LogWarning(Execute := _Warning, Arg0 := _Name, Arg1 := _Description, Arg2 := '', EventEntry := M_Warnings(), Clear := NOT _Warning, Message := Control.Outputs.WarningMessage);

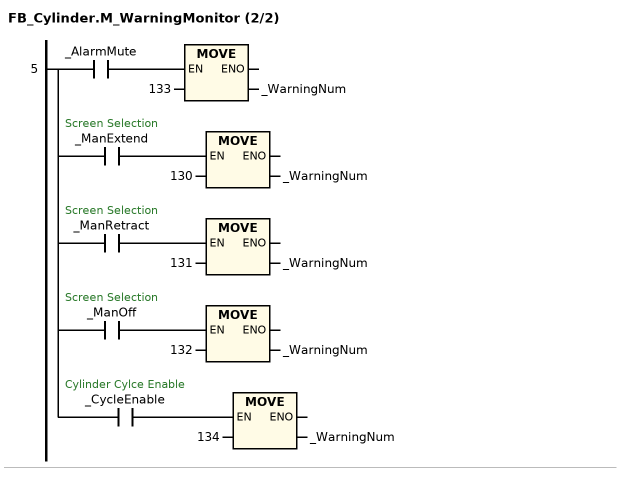
// NETWORK 5
//   _ManExtend: Screen Selection
//   _ManRetract: Screen Selection
//   _ManOff: Screen Selection
//   _CycleEnable: Cylinder Cylce Enable
_w3 := _AlarmMute;
IF _w3 THEN _WarningNum := 133; END_IF
_w4 := _ManExtend;
IF _w4 THEN _WarningNum := 130; END_IF
_w5 := _ManRetract;
IF _w5 THEN _WarningNum := 131; END_IF
_w6 := _ManOff;
IF _w6 THEN _WarningNum := 132; END_IF
_w7 := _CycleEnable;
IF _w7 THEN _WarningNum := 134; END_IF
(* _w3 OR _w4 OR _w5 OR _w6 OR _w7; result not used *)
END_METHOD

METHOD PRIVATE M_Warnings : TcEventEntry
VAR_INPUT
END_VAR
CASE _WarningNum OF
	130: M_Warnings:= TC_Events.TcCylinder.W_130;//Manual Extend Enabled	
	131: M_Warnings:= TC_Events.TcCylinder.W_131;//Manual Retract Enabled		
	132: M_Warnings:= TC_Events.TcCylinder.W_132;//Manual OFF Enabled
	133: M_Warnings:= TC_Events.TcCylinder.W_133;//Alarm Mute Active
	134: M_Warnings:= TC_Events.TcCylinder.W_134;//Cylinder Cycling Enabled					
ELSE
	M_Warnings:=  TC_Events.TcCylinder.W_Undefined;
END_CASE
END_METHOD

{attribute 'monitoring' := 'variable'}
PROPERTY PUBLIC ManExtend : Bool
GET
ManExtend := _ManExtend;
END_GET
SET
_ManExtend := ManExtend;
END_SET
END_PROPERTY

{attribute 'monitoring' := 'variable'}
PROPERTY PUBLIC ManOff : Bool
GET
ManOff := _ManOff;
END_GET
SET
_ManOff := ManOff;
END_SET
END_PROPERTY

{attribute 'monitoring' := 'variable'}
PROPERTY PUBLIC ManRetract : Bool
GET
ManRetract := _ManRetract;
END_GET
SET
_ManRetract := ManRetract;
END_SET
END_PROPERTY

{attribute 'monitoring' := 'variable'}
PROPERTY PUBLIC Name : String[15]
GET
Name := _Name;
END_GET
SET
_Name := Name;
END_SET
END_PROPERTY

{attribute 'monitoring' := 'variable'}
PROPERTY PUBLIC ReedFaultTime_ET : real
GET
ReedFaultTime_ET := _ReedFaultTime_ET;
END_GET
END_PROPERTY

{attribute 'monitoring' := 'variable'}
PROPERTY PUBLIC ReedFaultTime_PT : real
GET
ReedFaultTime_PT := _ReedFaultTime_PT;
END_GET
SET
_ReedFaultTime_PT := ReedFaultTime_PT;
END_SET
END_PROPERTY

{attribute 'monitoring' := 'variable'}
PROPERTY PUBLIC RetractReed : Bool
GET
RetractReed := _RetractReed;
END_GET
END_PROPERTY

{attribute 'monitoring' := 'variable'}
PROPERTY PUBLIC RetractReed1 : Bool
GET
RetractReed1 := _RetractReed1;
END_GET
SET // PUBLIC
_RetractReed1 := RetractReed1;
END_SET
END_PROPERTY

{attribute 'monitoring' := 'variable'}
PROPERTY PUBLIC RetractSol : Bool
GET
RetractSol := _RetractSol;
END_GET
END_PROPERTY

{attribute 'monitoring' := 'variable'}
PROPERTY PUBLIC RtFaultTime_ET : real
GET
RtFaultTime_ET := _RtFaultTime_ET;
END_GET
END_PROPERTY

{attribute 'monitoring' := 'variable'}
PROPERTY PUBLIC RtFaultTime_PT : real
GET
RtFaultTime_PT := _RtFaultTime_PT;
END_GET
SET
_RtFaultTime_PT := RtFaultTime_PT;
END_SET
END_PROPERTY

{attribute 'monitoring' := 'variable'}
PROPERTY PUBLIC StandbyReset : Bool
GET
StandbyReset := _ForceOff;
END_GET
SET
_ForceOff := StandbyReset;
END_SET
END_PROPERTY

PROPERTY PUBLIC Variables : REFERENCE TO ARRAY[0..9] OF ST_Variable
GET
Variables REF= _Variables;
END_GET
END_PROPERTY

{attribute 'monitoring' := 'variable'}
PROPERTY PUBLIC Warning : Bool
GET
Warning := _Warning;
END_GET
END_PROPERTY

END_FUNCTION_BLOCK

(* stored: Version 1.1.0.1, ProductVersion 3.1.4024.3
   POU FB_Cylinder: Id {040f7626-abee-4cfc-b764-c2362300adf8}, SpecialFunc None
   Property Alarm: Id {aa7355c0-70e6-4d9e-990a-718317068b89}
   Get Get: Id {a29a8b52-51d0-4c92-8ced-b819fae42695}
   Property AlarmMute: Id {2ad25553-3d62-49ac-90bc-f3f123ac989d}
   Set Set: Id {2b904e37-80b7-4c49-94fd-c0a0a6294205}
   Property AutoExtend: Id {3c35040c-8a56-44ef-982f-40c8d56c4959}
   Set Set: Id {34b10675-203e-4eac-a324-8ae20ab3c368}
   Property AutoRetract: Id {34bb80e2-27ea-445c-9ac7-cb05d424d55b}
   Set Set: Id {8f2e243c-25ca-4303-8fea-5199bb1a540d}
   Property CycleExtTime_PT: Id {8e5506d4-c937-4609-a055-8414d1eb5a8f}
   Get Get: Id {ba0ec80b-00a7-4a9d-87ca-0229df434d89}
   Set Set: Id {4459cbdd-3564-47b7-99af-ac3d03c014c6}
   Property CycleRetTime_PT: Id {f1d6539a-6a9c-4962-a5b3-ab1476b49414}
   Get Get: Id {c9f83a8d-2e50-4ffe-b609-8ae73f7785c6}
   Set Set: Id {d8d6439f-8163-454b-9dc3-95d7e5835080}
   Property Description: Id {e343646c-9680-4230-82a8-3ada12f84913}
   Get Get: Id {6338d223-d5d4-4cfe-89b0-69e5a47ebeeb}
   Set Set: Id {ae13851c-ad40-43d0-a1c6-4cc720f5c163}
   Property ExFaultTime_ET: Id {2941d210-3277-4e5e-98f3-e0c8838a17a4}
   Get Get: Id {aae938cf-c91e-4c78-9e90-1cdf4aa4e38a}
   Property ExFaultTime_PT: Id {806726ce-07d4-4856-be78-b204af106e55}
   Get Get: Id {b32c017d-5d52-41d7-9c6a-7f905e25f9a5}
   Set Set: Id {3aaad3d2-1197-4d52-af3c-6146145aee5e}
   Property ExtendReed: Id {6d62f9e1-1ac0-43f9-957b-ba1d04ab3be0}
   Get Get: Id {e303c26c-9208-41bd-842b-e5b22cd0b102}
   Property ExtendReed1: Id {de3ee508-0361-421b-8fef-3176dce60968}
   Get Get: Id {658252ac-6193-45e0-b718-1da4241cdefd}
   Set Set: Id {226a20fc-6333-4232-90b8-24eee5426195}
   Property ExtendSol: Id {b7f12936-ee04-41aa-b24a-30ccb56d39ee}
   Get Get: Id {f1d2b2ee-8d3b-456f-9d7e-dd50909d611e}
   Property ForceExtend: Id {678eb844-580f-42b4-8cc8-563b42b14543}
   Get Get: Id {e162b18d-2179-431b-a350-3c4d4014a20a}
   Set Set: Id {d52ec8b9-84c4-4dff-9fce-f0e0d3226eeb}
   Property ForceRetract: Id {4d911913-9ee7-49a2-8d48-71d3a767d1a7}
   Get Get: Id {4dcbeb5f-f44f-4ffa-aecd-148e1d1fc52f}
   Set Set: Id {8942d7f7-8705-40aa-8f0b-d26f56452d0b}
   Method M_AlarmMonitor: Id {a93b58bb-b9d8-4428-bb70-a7336d50c0ad}
   Method M_Alarms: Id {2b88edcd-60b2-4162-9353-c3fa5545a8c0}
   Method M_CountsReset: Id {69db508f-4965-46a1-911b-9dae6524fdba}
   Method M_Extend: Id {01479100-b531-468b-ae63-fe45f1f9a64a}
   Method M_ExtendFault: Id {3b4447b6-ef42-4c91-827d-160d2d9edcc8}
   Method M_ReedControl: Id {dbab9411-29f2-443f-8869-82f22f0cf0bc}
   Method M_ReedFault: Id {5889435f-84e4-403d-9fa1-bdf590a7cc54}
   Method M_Retract: Id {721983f6-a5c4-482a-a952-034cfd7e933f}
   Method M_RetractFault: Id {75d62904-2d5e-4f3f-8ed7-418901d8f8a8}
   Method M_TestCycle: Id {3a802ced-e391-4eb9-aefa-02149cdcb112}
   Method M_TypeConfig: Id {b5fca9c2-b7a3-47ae-bab1-9c415d5e1de5}
   Method M_UnlatchManuals: Id {06c3250c-f588-4700-9f47-f7d462fd7055}
   Method M_WarningMonitor: Id {51e8a362-4f81-4e66-9587-86834b8ce846}
   Method M_Warnings: Id {51379eb8-ec42-42c4-8675-02075695e4c0}
   Property ManExtend: Id {ead1efc0-81fb-4742-bf2d-2498287c38e0}
   Get Get: Id {74bb1bf1-5ac8-41b8-9838-7f62f19c9e73}
   Set Set: Id {da63f43e-8187-4526-9dec-b27179bf960f}
   Property ManOff: Id {646a9dc6-3de2-4f43-8c81-83ea5921ef36}
   Get Get: Id {f17905ba-590b-463e-aa12-2c2086f88fb5}
   Set Set: Id {b55bad23-76fd-45be-b691-d7aad0add3a9}
   Property ManRetract: Id {ff02391e-f7a1-49cf-9599-6102711cbe35}
   Get Get: Id {9c5ac358-e833-44d3-9a3f-b4f1ae638c5c}
   Set Set: Id {afefae5c-7fca-41a4-8bdb-0ccd5cb27b69}
   Property Name: Id {4f9ce7ee-2f02-47d9-9d3f-4cde66ce5608}
   Get Get: Id {edd0fca4-413b-4f93-94d3-da96ec791e3f}
   Set Set: Id {5800a42e-600b-4338-a451-9bed6021a809}
   Property ReedFaultTime_ET: Id {9a2f3d76-3838-4705-817e-2e1b95730228}
   Get Get: Id {8f8af83c-6015-46ea-839f-b5c22a9c5cb8}
   Property ReedFaultTime_PT: Id {de5b9de3-e1da-4f89-a396-61ab09c9e2e3}
   Get Get: Id {892c8da1-cec3-48d9-abc6-d62607d4bc6e}
   Set Set: Id {8e4001e4-fc20-4362-a8e2-584831b569ef}
   Property RetractReed: Id {6b4ed962-d69a-4dcd-ae19-f71407a7b502}
   Get Get: Id {4eb2dfdf-b899-49fc-b24f-01b67d2ded42}
   Property RetractReed1: Id {fc8cba56-4cc4-4809-aafc-e61e653c3439}
   Get Get: Id {6134e733-fbaa-464b-959a-4a46a47a4522}
   Set Set: Id {b9ae1a5d-68b6-4dd7-ab07-4a8962b84142}
   Property RetractSol: Id {3c724451-82da-4d8a-ae3d-e08c8b46625d}
   Get Get: Id {878db4b6-7290-4fa4-b8a8-4fc29ec5f6f7}
   Property RtFaultTime_ET: Id {a7c391b1-d2e0-4a81-ab67-2396243380aa}
   Get Get: Id {5a403c12-6da4-462d-ba52-ec6a58613d19}
   Property RtFaultTime_PT: Id {99758617-e5a8-4b23-bae8-7ca2a5ed7382}
   Get Get: Id {73a5e43e-caf5-478e-80be-8c1c5be08f10}
   Set Set: Id {0e4d98c4-91df-44e3-b368-d0ef45cf2983}
   Property StandbyReset: Id {d15bce0f-9f14-4f03-9a65-aa0533b69176}
   Get Get: Id {34ad9471-8529-43b6-9ca4-fccb9ca7ead7}
   Set Set: Id {9574b754-fc74-490c-a5a3-8bd9cdded82a}
   Property Variables: Id {23bbba2c-505f-4e10-a283-89a2aa826312}
   Get Get: Id {edc1da4d-a5f5-4cfa-a7d6-e75f588d6886}
   Property Warning: Id {427b2fe8-d18d-44aa-88fb-7fb59e4eddda}
   Get Get: Id {7e0cd938-e806-40ce-9594-0b4ffabc5b74} *)
